{attribute 'qualified_only'}
{attribute 'strict'}
TYPE E_COE_PTP_STATE :
(   
	UNKNOWN := -1,
	LISTENING := 4,
	SLAVE := 9
);
END_TYPE

(* stored: Version 1.1.0.1, ProductVersion 3.1.4022.12
   DUT E_COE_PTP_STATE: Id {7f82ead7-229e-445c-88f5-4898f7366c67} *)
